Universal Robots URScript: 07_Force_measurement_01.script

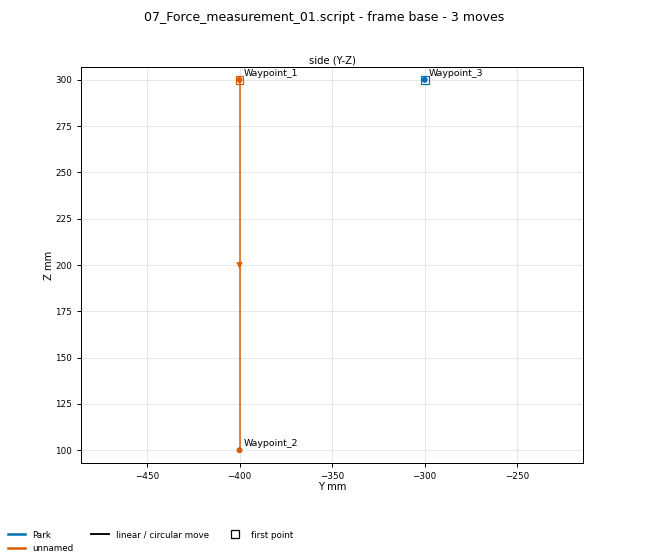
[picture p0: tool path of 07_Force_measurement_01.script in frame base, 3 of 3 moves have a stored position in this frame; points joined in program order, loops and branches not executed]
def unnamed():
  step_count_77154f07_a93b_4dac_9cdc_12584ce3cc98 = 0.0
  thread Step_Counter_Thread_65f37794_2095_4b5c_a568_ff3977c41b84():
    while (True):
      step_count_77154f07_a93b_4dac_9cdc_12584ce3cc98 = step_count_77154f07_a93b_4dac_9cdc_12584ce3cc98 + 1.0
      sync()
    end
  end
  run Step_Counter_Thread_65f37794_2095_4b5c_a568_ff3977c41b84()
  set_tcp(p[0.0,0.0,0.0,0.0,0.0,0.0])
  set_payload(0.0)
  set_standard_analog_input_domain(0, 1)
  set_standard_analog_input_domain(1, 1)
  set_tool_analog_input_domain(0, 1)
  set_tool_analog_input_domain(1, 1)
  set_analog_outputdomain(0, 0)
  set_analog_outputdomain(1, 0)
  set_input_actions_to_default()
  set_gravity([0.0, 0.0, 9.82])
  set_tool_communication(False, 115200, 0, 1, 1.5, 3.5)
  set_tool_output_mode(0)
  set_tool_digital_output_mode(0, 1)
  set_tool_digital_output_mode(1, 1)
  set_tool_voltage(0)
  set_safety_mode_transition_hardness(1)
  global i_count=5
  global Waypoint_1_p=p[-.000000000021, -.400000000005, .299999999985, .000000003497, 3.141592653590, .000000001105]
  global Waypoint_1_q=[-1.2310478043488384, -1.405522179080525, -2.2189438958375503, -1.087922905930153, 1.5707963268097895, 0.3397485248773866]
  global Waypoint_2_p=p[-.000000000021, -.400000000005, .099999999890, .000000003497, 3.141592653590, .000000001105]
  global Waypoint_2_q=[-1.2310478044613866, -1.8956434733253467, -2.4468407926978353, -0.3699047148199872, 1.5707963268241036, 0.33974852476484524]
  global Waypoint_3_p=p[-.000000000021, -.299999999964, .300000000073, .000000003497, 3.141592653590, .000000001105]
  global Waypoint_3_q=[-1.1103663660542393, -1.0871644383714179, -2.417142038724915, -1.2080825037136913, 1.5707963269025116, 0.46042996317199103]
  def Park():
    $ 10 "Park" "noBreak"
    $ 11 "MoveL"
    $ 12 "Waypoint_3" "breakAfter"
    movel(Waypoint_3_p, a=1.2, v=0.25)
    $ 13 "Set DO[0]=Off"
    set_standard_digital_out(0, False)
    $ 14 "Wait: 3.0"
    sleep(3.0)
    $ 15 "Fmax≔0"
    global Fmax=0
  end
  $ 19 "Thread_1"
  thread Thread_1():
    while (True):
      $ 20 "Wait: 0.01"
      sleep(0.01)
      $ 21 "ForceValue≔force()"
      global ForceValue= force ()
    end
  end
  threadId_Thread_1 = run Thread_1()
  thread EventThread():
    while (True):
      if (ForceValue>40):
        $ 17 "Fmax≔1"
        global Fmax=1
        $ 18 "Set DO[0]=On"
        set_standard_digital_out(0, True)
      end
      sync()
    end
  end
  eventThread = run EventThread()
  while (True):
    $ 2 "Robot Program"
    $ 3 "MoveL"
    $ 4 "Waypoint_1" "breakAfter"
    movel(Waypoint_1_p, a=1.2, v=0.25)
    $ 5 "Force"
    sleep(0.02)
    zero_ftsensor()
    force_mode(p[0.0,0.0,0.0,0.0,0.0,0.0], [0, 0, 1, 0, 0, 0], [0.0, 0.0, 10.0, 0.0, 0.0, 0.0], 2, [0.1, 0.1, 0.15, 0.3490658503988659, 0.3490658503988659, 0.3490658503988659])
    $ 6 "MoveL" "noBreak"
    $ 7 "Waypoint_2" "noBreak"
    movel(Waypoint_2_p, a=1.2, v=0.25)
    end_force_mode()
    stopl(5.0)
    $ 8 "If Fmax≟1"
    if (Fmax == 1):
      $ 9 "Call Park"
      Park()
    end
  end
end
